FUNCTION_BLOCK FB_XmlPersistentEventStorage IMPLEMENTS I_PersistentEventStorage
VAR_INPUT
END_VAR
VAR_OUTPUT
END_VAR
VAR
END_VAR

{warning 'add method implementation '}
METHOD StoreEvent
VAR_INPUT
	stEvent	: ST_Event;
END_VAR
// Here is there XML-Writing is supposed to be done
//Were is where the FB_XmlPersistentEventStorage se debe implementar el codigo aqui.
END_METHOD

END_FUNCTION_BLOCK

(* stored: Version 1.1.0.1, ProductVersion 3.1.4024.12
   POU FB_XmlPersistentEventStorage: Id {415bbc5a-7ea8-4617-896a-299e0238dbff}, SpecialFunc None
   Method StoreEvent: Id {84c531b4-e2f0-45fd-8194-f1da4a2ee6dc} *)
